INTERFACE I_ActuatorUpDown EXTENDS I_ActuatorBase

{attribute 'monitoring' := 'call'}
PROPERTY public downOk : BOOL
GET
END_GET
END_PROPERTY

METHOD public moveDown : BOOL
VAR_INPUT
END_VAR
END_METHOD

METHOD public moveUp : BOOL
VAR_INPUT
END_VAR
END_METHOD

{attribute 'monitoring' := 'call'}
PROPERTY public upOK : BOOL
GET
END_GET
END_PROPERTY

END_INTERFACE

(* stored: Version 1.1.0.1, ProductVersion 3.1.4024.3
   Itf I_ActuatorUpDown: Id {c6a6a5fa-2410-408f-9be1-da95dab0841f}
   Property downOk: Id {26256a76-3c63-477a-8a4a-f1a82805d139}
   Get Get: Id {000d82fd-63c8-4741-a741-eb4a4b4cbae7}
   Method moveDown: Id {06ade7e5-25a6-4c23-aee7-cde9e9fdf274}
   Method moveUp: Id {b7ebaa68-88fe-40af-b5f9-af58f000bcc4}
   Property upOK: Id {597b27d4-7aa3-47b6-931b-21e158fd7587}
   Get Get: Id {6af2f25a-7886-4521-bfa7-c44ffb354d7a} *)
